FUNCTION_BLOCK PS_PackML_StateMachine_Auto
VAR_INPUT
	Start					:	BOOL;
	Hold					:	BOOL;
	UnHold					:	BOOL;
	Suspend					:	BOOL;
	UnSuspend				:	BOOL;
	Abort					:	BOOL;
	Stop					:	BOOL;
	Complete				:	BOOL;
	Clear					:	BOOL;
	Reset					:	BOOL;
	StateComplete			:	BOOL;
END_VAR
VAR_OUTPUT
	Status					:	WORD;
	// Transient states
	ST_Starting				:	BOOL;
	ST_Completing			:	BOOL;
	ST_Resetting			:	BOOL;
	ST_Holding				:	BOOL;
	ST_UnHolding			:	BOOL;
	ST_Suspending			:	BOOL;
	ST_UnSuspending			:	BOOL;
	ST_Clearing				:	BOOL;
	ST_Stopping				:	BOOL;
	ST_Aborting				:	BOOL;
	// Final states
	ST_Execute				:	BOOL;
	ST_Complete				:	BOOL;
	ST_Idle					:	BOOL;
	ST_Held					:	BOOL;
	ST_Suspended			:	BOOL;
	ST_Stopped				:	BOOL;
	ST_Aborted				:	BOOL;
	
	Error					:	BOOL;
	ErrorID					:	DWORD;
	ePMLState				:	E_PMLState	:=	E_PMLState.IDLE;
END_VAR
VAR
	ePMLStatePrev			:	E_PMLState;
	bStateChange			:	BOOL;
	bStateCompletePrev		:	BOOL;
END_VAR

	// Check for E_PMLState change
	IF ePMLStatePrev <> ePMLState THEN
		ePMLStatePrev	:=	ePMLState;
		bStateChange	:=	TRUE;
	ELSE
		bStateChange	:=	FALSE;
	END_IF
	
	// change to new state if requested
	CASE ePMLState OF
		E_PMLState.UNDEFINED:
			IF bStateChange	THEN
				ST_Starting				:=	FALSE;
				ST_Completing			:=	FALSE;
				ST_Resetting			:=	FALSE;
				ST_Holding				:=	FALSE;
				ST_UnHolding			:=	FALSE;
				ST_Suspending			:=	FALSE;
				ST_UnSuspending			:=	FALSE;
				ST_Clearing				:=	FALSE;
				ST_Stopping				:=	FALSE;
				ST_Aborting				:=	FALSE;
				
				ST_Execute				:=	FALSE;
				ST_Complete				:=	FALSE;
				ST_Idle					:=	FALSE;
				ST_Held					:=	FALSE;
				ST_Suspended			:=	FALSE;
				ST_Stopped				:=	FALSE;
				ST_Aborted				:=	FALSE;
			END_IF
			
			IF Abort THEN
				ePMLState				:=	E_PMLState.ABORTING;
				ST_Aborting				:=	TRUE;
			ELSIF Stop THEN
				ePMLState				:=	E_PMLState.STOPPING;
				ST_Stopping				:=	TRUE;				
			END_IF
		E_PMLState.IDLE:
			IF bStateChange	THEN
				ST_Starting				:=	FALSE;
				ST_Completing			:=	FALSE;
				ST_Resetting			:=	FALSE;
				ST_Holding				:=	FALSE;
				ST_UnHolding			:=	FALSE;
				ST_Suspending			:=	FALSE;
				ST_UnSuspending			:=	FALSE;
				ST_Clearing				:=	FALSE;
				ST_Stopping				:=	FALSE;
				ST_Aborting				:=	FALSE;
				
				ST_Execute				:=	FALSE;
				ST_Complete				:=	FALSE;
				ST_Idle					:=	TRUE;
				ST_Held					:=	FALSE;
				ST_Suspended			:=	FALSE;
				ST_Stopped				:=	FALSE;
				ST_Aborted				:=	FALSE;
			END_IF
			
			IF Abort THEN
				ePMLState				:=	E_PMLState.ABORTING;
				ST_IDLE					:=	FALSE;
				ST_Aborting				:=	TRUE;
			ELSIF Stop THEN
				ePMLState				:=	E_PMLState.STOPPING;
				ST_IDLE					:=	FALSE;
				ST_Stopping				:=	TRUE;
			ELSIF Start THEN
				ePMLState				:=	E_PMLState.STARTING;
				ST_IDLE					:=	FALSE;
				ST_Starting				:=	TRUE;								
			END_IF

		E_PMLState.STARTING:
			IF bStateChange	THEN
				ST_Starting				:=	TRUE;
				ST_Completing			:=	FALSE;
				ST_Resetting			:=	FALSE;
				ST_Holding				:=	FALSE;
				ST_UnHolding			:=	FALSE;
				ST_Suspending			:=	FALSE;
				ST_UnSuspending			:=	FALSE;
				ST_Clearing				:=	FALSE;
				ST_Stopping				:=	FALSE;
				ST_Aborting				:=	FALSE;
				
				ST_Execute				:=	FALSE;
				ST_Complete				:=	FALSE;
				ST_Idle					:=	FALSE;
				ST_Held					:=	FALSE;
				ST_Suspended			:=	FALSE;
				ST_Stopped				:=	FALSE;
				ST_Aborted				:=	FALSE;
			END_IF
			
			IF Abort THEN
				ePMLState				:=	E_PMLState.ABORTING;
				ST_Starting				:=	FALSE;
				ST_Aborting				:=	TRUE;
			ELSIF Stop THEN
				ePMLState				:=	E_PMLState.STOPPING;
				ST_Starting				:=	FALSE;
				ST_Stopping				:=	TRUE;
			ELSIF StateComplete AND NOT bStateCompletePrev THEN
				ePMLState				:=	E_PMLState.EXECUTE;
				bStateCompletePrev		:=	StateComplete;
				ST_Starting				:=	FALSE;
				ST_Execute				:=	TRUE;								
			END_IF

		E_PMLState.EXECUTE:
			IF bStateChange	THEN
				ST_Starting				:=	FALSE;
				ST_Completing			:=	FALSE;
				ST_Resetting			:=	FALSE;
				ST_Holding				:=	FALSE;
				ST_UnHolding			:=	FALSE;
				ST_Suspending			:=	FALSE;
				ST_UnSuspending			:=	FALSE;
				ST_Clearing				:=	FALSE;
				ST_Stopping				:=	FALSE;
				ST_Aborting				:=	FALSE;
				
				ST_Execute				:=	TRUE;
				ST_Complete				:=	FALSE;
				ST_Idle					:=	FALSE;
				ST_Held					:=	FALSE;
				ST_Suspended			:=	FALSE;
				ST_Stopped				:=	FALSE;
				ST_Aborted				:=	FALSE;
			END_IF
			
			IF Abort THEN
				ePMLState				:=	E_PMLState.ABORTING;
				ST_Execute				:=	FALSE;
				ST_Aborting				:=	TRUE;
			ELSIF Stop THEN
				ePMLState				:=	E_PMLState.STOPPING;
				ST_Execute				:=	FALSE;
				ST_Stopping				:=	TRUE;
			ELSIF Hold THEN
				ePMLState				:=	E_PMLState.HOLDING;
				ST_Execute				:=	FALSE;
				ST_Holding				:=	TRUE;
			ELSIF Suspend THEN
				ePMLState				:=	E_PMLState.SUSPENDING;
				ST_Execute				:=	FALSE;
				ST_Suspending			:=	TRUE;
			ELSIF Complete THEN
				ePMLState				:=	E_PMLState.COMPLETING;
				ST_Execute				:=	FALSE;
				ST_Completing			:=	TRUE;	
			END_IF

		E_PMLState.COMPLETING:
			IF bStateChange	THEN
				ST_Starting				:=	FALSE;
				ST_Completing			:=	TRUE;
				ST_Resetting			:=	FALSE;
				ST_Holding				:=	FALSE;
				ST_UnHolding			:=	FALSE;
				ST_Suspending			:=	FALSE;
				ST_UnSuspending			:=	FALSE;
				ST_Clearing				:=	FALSE;
				ST_Stopping				:=	FALSE;
				ST_Aborting				:=	FALSE;
				
				ST_Execute				:=	FALSE;
				ST_Complete				:=	FALSE;
				ST_Idle					:=	FALSE;
				ST_Held					:=	FALSE;
				ST_Suspended			:=	FALSE;
				ST_Stopped				:=	FALSE;
				ST_Aborted				:=	FALSE;
			END_IF
			
			IF Abort THEN
				ePMLState				:=	E_PMLState.ABORTING;
				ST_Completing			:=	FALSE;
				ST_Aborting				:=	TRUE;
			ELSIF Stop THEN
				ePMLState				:=	E_PMLState.STOPPING;
				ST_Completing			:=	FALSE;
				ST_Stopping				:=	TRUE;
			ELSIF StateComplete AND NOT bStateCompletePrev THEN
				ePMLState				:=	E_PMLState.COMPLETE;
				bStateCompletePrev		:=	StateComplete;
				ST_Completing			:=	FALSE;
				ST_Complete				:=	TRUE;								
			END_IF
			
		E_PMLState.COMPLETE:
			IF bStateChange	THEN
				ST_Starting				:=	FALSE;
				ST_Completing			:=	FALSE;
				ST_Resetting			:=	FALSE;
				ST_Holding				:=	FALSE;
				ST_UnHolding			:=	FALSE;
				ST_Suspending			:=	FALSE;
				ST_UnSuspending			:=	FALSE;
				ST_Clearing				:=	FALSE;
				ST_Stopping				:=	FALSE;
				ST_Aborting				:=	FALSE;
				
				ST_Execute				:=	FALSE;
				ST_Complete				:=	TRUE;
				ST_Idle					:=	FALSE;
				ST_Held					:=	FALSE;
				ST_Suspended			:=	FALSE;
				ST_Stopped				:=	FALSE;
				ST_Aborted				:=	FALSE;
			END_IF
			
			IF Abort THEN
				ePMLState				:=	E_PMLState.ABORTING;
				ST_Complete				:=	FALSE;
				ST_Aborting				:=	TRUE;
			ELSIF Stop THEN
				ePMLState				:=	E_PMLState.STOPPING;
				ST_Complete				:=	FALSE;
				ST_Stopping				:=	TRUE;
			ELSIF Reset THEN
				ePMLState				:=	E_PMLState.RESETTING;
				ST_Complete				:=	FALSE;
				ST_Resetting			:=	TRUE;
			END_IF

		E_PMLState.RESETTING:
			IF bStateChange	THEN
				ST_Starting				:=	FALSE;
				ST_Completing			:=	FALSE;
				ST_Resetting			:=	TRUE;
				ST_Holding				:=	FALSE;
				ST_UnHolding			:=	FALSE;
				ST_Suspending			:=	FALSE;
				ST_UnSuspending			:=	FALSE;
				ST_Clearing				:=	FALSE;
				ST_Stopping				:=	FALSE;
				ST_Aborting				:=	FALSE;
				
				ST_Execute				:=	FALSE;
				ST_Complete				:=	FALSE;
				ST_Idle					:=	FALSE;
				ST_Held					:=	FALSE;
				ST_Suspended			:=	FALSE;
				ST_Stopped				:=	FALSE;
				ST_Aborted				:=	FALSE;
			END_IF
			
			IF Abort THEN
				ePMLState				:=	E_PMLState.ABORTING;
				ST_Resetting			:=	FALSE;
				ST_Aborting				:=	TRUE;
			ELSIF Stop THEN
				ePMLState				:=	E_PMLState.STOPPING;
				ST_Resetting			:=	FALSE;
				ST_Stopping				:=	TRUE;
			ELSIF StateComplete AND NOT bStateCompletePrev THEN
				ePMLState				:=	E_PMLState.IDLE;
				bStateCompletePrev		:=	StateComplete;
				ST_Resetting			:=	FALSE;
				ST_Idle					:=	TRUE;								
			END_IF
		
		E_PMLState.HOLDING:
			IF bStateChange	THEN
				ST_Starting				:=	FALSE;
				ST_Completing			:=	FALSE;
				ST_Resetting			:=	FALSE;
				ST_Holding				:=	TRUE;
				ST_UnHolding			:=	FALSE;
				ST_Suspending			:=	FALSE;
				ST_UnSuspending			:=	FALSE;
				ST_Clearing				:=	FALSE;
				ST_Stopping				:=	FALSE;
				ST_Aborting				:=	FALSE;
				
				ST_Execute				:=	FALSE;
				ST_Complete				:=	FALSE;
				ST_Idle					:=	FALSE;
				ST_Held					:=	FALSE;
				ST_Suspended			:=	FALSE;
				ST_Stopped				:=	FALSE;
				ST_Aborted				:=	FALSE;
			END_IF
			
			IF Abort THEN
				ePMLState				:=	E_PMLState.ABORTING;
				ST_Holding				:=	FALSE;
				ST_Aborting				:=	TRUE;
			ELSIF Stop THEN
				ePMLState				:=	E_PMLState.STOPPING;
				ST_Holding				:=	FALSE;
				ST_Stopping				:=	TRUE;
			ELSIF StateComplete AND NOT bStateCompletePrev THEN
				ePMLState				:=	E_PMLState.HELD;
				bStateCompletePrev		:=	StateComplete;
				ST_Holding				:=	FALSE;
				ST_Held					:=	TRUE;								
			END_IF
			
		E_PMLState.HELD:
			IF bStateChange	THEN
				ST_Starting				:=	FALSE;
				ST_Completing			:=	FALSE;
				ST_Resetting			:=	FALSE;
				ST_Holding				:=	FALSE;
				ST_UnHolding			:=	FALSE;
				ST_Suspending			:=	FALSE;
				ST_UnSuspending			:=	FALSE;
				ST_Clearing				:=	FALSE;
				ST_Stopping				:=	FALSE;
				ST_Aborting				:=	FALSE;
				
				ST_Execute				:=	FALSE;
				ST_Complete				:=	FALSE;
				ST_Idle					:=	FALSE;
				ST_Held					:=	TRUE;
				ST_Suspended			:=	FALSE;
				ST_Stopped				:=	FALSE;
				ST_Aborted				:=	FALSE;
			END_IF
			
			IF Abort THEN
				ePMLState				:=	E_PMLState.ABORTING;
				ST_Held					:=	FALSE;
				ST_Aborting				:=	TRUE;
			ELSIF Stop THEN
				ePMLState				:=	E_PMLState.STOPPING;
				ST_Held					:=	FALSE;
				ST_Stopping				:=	TRUE;
			ELSIF UnHold THEN
				ePMLState				:=	E_PMLState.UNHOLDING;
				ST_Held					:=	FALSE;
				ST_UnHolding			:=	TRUE;
			END_IF

		E_PMLState.UNHOLDING:	
			IF bStateChange	THEN
				ST_Starting				:=	FALSE;
				ST_Completing			:=	FALSE;
				ST_Resetting			:=	FALSE;
				ST_Holding				:=	FALSE;
				ST_UnHolding			:=	TRUE;
				ST_Suspending			:=	FALSE;
				ST_UnSuspending			:=	FALSE;
				ST_Clearing				:=	FALSE;
				ST_Stopping				:=	FALSE;
				ST_Aborting				:=	FALSE;
				
				ST_Execute				:=	FALSE;
				ST_Complete				:=	FALSE;
				ST_Idle					:=	FALSE;
				ST_Held					:=	FALSE;
				ST_Suspended			:=	FALSE;
				ST_Stopped				:=	FALSE;
				ST_Aborted				:=	FALSE;
			END_IF
			
			IF Abort THEN
				ePMLState				:=	E_PMLState.ABORTING;
				ST_UnHolding			:=	FALSE;
				ST_Aborting				:=	TRUE;
			ELSIF Stop THEN
				ePMLState				:=	E_PMLState.STOPPING;
				ST_UnHolding			:=	FALSE;
				ST_Stopping				:=	TRUE;
			ELSIF StateComplete AND NOT bStateCompletePrev THEN
				ePMLState				:=	E_PMLState.EXECUTE;
				bStateCompletePrev		:=	StateComplete;
				ST_UnHolding			:=	FALSE;
				ST_Execute				:=	TRUE;								
			END_IF
			
		E_PMLState.SUSPENDING:
			IF bStateChange	THEN
				ST_Starting				:=	FALSE;
				ST_Completing			:=	FALSE;
				ST_Resetting			:=	FALSE;
				ST_Holding				:=	FALSE;
				ST_UnHolding			:=	FALSE;
				ST_Suspending			:=	TRUE;
				ST_UnSuspending			:=	FALSE;
				ST_Clearing				:=	FALSE;
				ST_Stopping				:=	FALSE;
				ST_Aborting				:=	FALSE;
				
				ST_Execute				:=	FALSE;
				ST_Complete				:=	FALSE;
				ST_Idle					:=	FALSE;
				ST_Held					:=	FALSE;
				ST_Suspended			:=	FALSE;
				ST_Stopped				:=	FALSE;
				ST_Aborted				:=	FALSE;
			END_IF
			
			IF Abort THEN
				ePMLState				:=	E_PMLState.ABORTING;
				ST_Suspending			:=	FALSE;
				ST_Aborting				:=	TRUE;
			ELSIF Stop THEN
				ePMLState				:=	E_PMLState.STOPPING;
				ST_Suspending			:=	FALSE;
				ST_Stopping				:=	TRUE;
			ELSIF StateComplete AND NOT bStateCompletePrev THEN
				ePMLState				:=	E_PMLState.SUSPENDED;
				bStateCompletePrev		:=	StateComplete;
				ST_Suspending			:=	FALSE;
				ST_Suspended			:=	TRUE;								
			END_IF
		
		E_PMLState.SUSPENDED:
			IF bStateChange	THEN
				ST_Starting				:=	FALSE;
				ST_Completing			:=	FALSE;
				ST_Resetting			:=	FALSE;
				ST_Holding				:=	FALSE;
				ST_UnHolding			:=	FALSE;
				ST_Suspending			:=	FALSE;
				ST_UnSuspending			:=	FALSE;
				ST_Clearing				:=	FALSE;
				ST_Stopping				:=	FALSE;
				ST_Aborting				:=	FALSE;
				
				ST_Execute				:=	FALSE;
				ST_Complete				:=	FALSE;
				ST_Idle					:=	FALSE;
				ST_Held					:=	FALSE;
				ST_Suspended			:=	TRUE;
				ST_Stopped				:=	FALSE;
				ST_Aborted				:=	FALSE;
			END_IF
			
			IF Abort THEN
				ePMLState				:=	E_PMLState.ABORTING;
				ST_Suspended			:=	FALSE;
				ST_Aborting				:=	TRUE;
			ELSIF Stop THEN
				ePMLState				:=	E_PMLState.STOPPING;
				ST_Suspended			:=	FALSE;
				ST_Stopping				:=	TRUE;
			ELSIF UnSuspend THEN
				ePMLState				:=	E_PMLState.UNSUSPENDING;
				ST_Suspended			:=	FALSE;
				ST_UnSuspending			:=	TRUE;
			END_IF

		E_PMLState.UNSUSPENDING:	
			IF bStateChange	THEN
				ST_Starting				:=	FALSE;
				ST_Completing			:=	FALSE;
				ST_Resetting			:=	FALSE;
				ST_Holding				:=	FALSE;
				ST_UnHolding			:=	FALSE;
				ST_Suspending			:=	FALSE;
				ST_UnSuspending			:=	TRUE;
				ST_Clearing				:=	FALSE;
				ST_Stopping				:=	FALSE;
				ST_Aborting				:=	FALSE;
				
				ST_Execute				:=	FALSE;
				ST_Complete				:=	FALSE;
				ST_Idle					:=	FALSE;
				ST_Held					:=	FALSE;
				ST_Suspended			:=	FALSE;
				ST_Stopped				:=	FALSE;
				ST_Aborted				:=	FALSE;
			END_IF
			
			IF Abort THEN
				ePMLState				:=	E_PMLState.ABORTING;
				ST_UnSuspending			:=	FALSE;
				ST_Aborting				:=	TRUE;
			ELSIF Stop THEN
				ePMLState				:=	E_PMLState.STOPPING;
				ST_UnSuspending			:=	FALSE;
				ST_Stopping				:=	TRUE;
			ELSIF StateComplete AND NOT bStateCompletePrev THEN
				ePMLState				:=	E_PMLState.EXECUTE;
				bStateCompletePrev		:=	StateComplete;
				ST_UnSuspending			:=	FALSE;
				ST_Execute				:=	TRUE;								
			END_IF
		
		E_PMLState.STOPPING:
			IF bStateChange	THEN
				ST_Starting				:=	FALSE;
				ST_Completing			:=	FALSE;
				ST_Resetting			:=	FALSE;
				ST_Holding				:=	FALSE;
				ST_UnHolding			:=	FALSE;
				ST_Suspending			:=	FALSE;
				ST_UnSuspending			:=	FALSE;
				ST_Clearing				:=	FALSE;
				ST_Stopping				:=	TRUE;
				ST_Aborting				:=	FALSE;
				
				ST_Execute				:=	FALSE;
				ST_Complete				:=	FALSE;
				ST_Idle					:=	FALSE;
				ST_Held					:=	FALSE;
				ST_Suspended			:=	FALSE;
				ST_Stopped				:=	FALSE;
				ST_Aborted				:=	FALSE;
			END_IF
			
			IF Abort THEN
				ePMLState				:=	E_PMLState.ABORTING;
				ST_Stopping				:=	FALSE;
				ST_Aborting				:=	TRUE;
			ELSIF StateComplete AND NOT bStateCompletePrev THEN
				ePMLState				:=	E_PMLState.STOPPED;
				bStateCompletePrev		:=	StateComplete;
				ST_Stopping				:=	FALSE;
				ST_Stopped				:=	TRUE;								
			END_IF

		E_PMLState.STOPPED:
			IF bStateChange	THEN
				ST_Starting				:=	FALSE;
				ST_Completing			:=	FALSE;
				ST_Resetting			:=	FALSE;
				ST_Holding				:=	FALSE;
				ST_UnHolding			:=	FALSE;
				ST_Suspending			:=	FALSE;
				ST_UnSuspending			:=	FALSE;
				ST_Clearing				:=	FALSE;
				ST_Stopping				:=	FALSE;
				ST_Aborting				:=	FALSE;
				
				ST_Execute				:=	FALSE;
				ST_Complete				:=	FALSE;
				ST_Idle					:=	FALSE;
				ST_Held					:=	FALSE;
				ST_Suspended			:=	FALSE;
				ST_Stopped				:=	TRUE;
				ST_Aborted				:=	FALSE;
			END_IF
			
			IF Abort THEN
				ePMLState				:=	E_PMLState.ABORTING;
				ST_Stopped				:=	FALSE;
				ST_Aborting				:=	TRUE;
			ELSIF Reset THEN
				ePMLState				:=	E_PMLState.RESETTING;
				ST_Stopped				:=	FALSE;
				ST_Resetting			:=	TRUE;
			END_IF
		
		E_PMLState.ABORTING:
			IF bStateChange	THEN
				ST_Starting				:=	FALSE;
				ST_Completing			:=	FALSE;
				ST_Resetting			:=	FALSE;
				ST_Holding				:=	FALSE;
				ST_UnHolding			:=	FALSE;
				ST_Suspending			:=	FALSE;
				ST_UnSuspending			:=	FALSE;
				ST_Clearing				:=	FALSE;
				ST_Stopping				:=	FALSE;
				ST_Aborting				:=	TRUE;
				
				ST_Execute				:=	FALSE;
				ST_Complete				:=	FALSE;
				ST_Idle					:=	FALSE;
				ST_Held					:=	FALSE;
				ST_Suspended			:=	FALSE;
				ST_Stopped				:=	FALSE;
				ST_Aborted				:=	FALSE;
			END_IF
			
			IF StateComplete AND NOT bStateCompletePrev THEN
				ePMLState				:=	E_PMLState.ABORTED;
				bStateCompletePrev		:=	StateComplete;
				ST_Aborting				:=	FALSE;
				ST_Aborted				:=	TRUE;								
			END_IF
			
		E_PMLState.ABORTED:
			IF bStateChange	THEN
				ST_Starting				:=	FALSE;
				ST_Completing			:=	FALSE;
				ST_Resetting			:=	FALSE;
				ST_Holding				:=	FALSE;
				ST_UnHolding			:=	FALSE;
				ST_Suspending			:=	FALSE;
				ST_UnSuspending			:=	FALSE;
				ST_Clearing				:=	FALSE;
				ST_Stopping				:=	FALSE;
				ST_Aborting				:=	FALSE;
				
				ST_Execute				:=	FALSE;
				ST_Complete				:=	FALSE;
				ST_Idle					:=	FALSE;
				ST_Held					:=	FALSE;
				ST_Suspended			:=	FALSE;
				ST_Stopped				:=	FALSE;
				ST_Aborted				:=	TRUE;
			END_IF
			
			IF Clear THEN
				ePMLState				:=	E_PMLState.CLEARING;
				ST_Aborted				:=	FALSE;
				ST_Clearing				:=	TRUE;
			END_IF
		
		E_PMLState.CLEARING:
			IF bStateChange	THEN
				ST_Starting				:=	FALSE;
				ST_Completing			:=	FALSE;
				ST_Resetting			:=	FALSE;
				ST_Holding				:=	FALSE;
				ST_UnHolding			:=	FALSE;
				ST_Suspending			:=	FALSE;
				ST_UnSuspending			:=	FALSE;
				ST_Clearing				:=	TRUE;
				ST_Stopping				:=	FALSE;
				ST_Aborting				:=	FALSE;
				
				ST_Execute				:=	FALSE;
				ST_Complete				:=	FALSE;
				ST_Idle					:=	FALSE;
				ST_Held					:=	FALSE;
				ST_Suspended			:=	FALSE;
				ST_Stopped				:=	FALSE;
				ST_Aborted				:=	FALSE;
			END_IF
			
			IF Abort THEN
				ePMLState				:=	E_PMLState.ABORTING;
				ST_Clearing				:=	FALSE;
				ST_Aborting				:=	TRUE;
			ELSIF Stop THEN
				ePMLState				:=	E_PMLState.STOPPING;
				ST_Clearing				:=	FALSE;
				ST_Stopping				:=	TRUE;
			ELSIF StateComplete AND NOT bStateCompletePrev THEN
				ePMLState				:=	E_PMLState.STOPPED;
				bStateCompletePrev		:=	StateComplete;
				ST_Clearing				:=	FALSE;
				ST_Stopped				:=	TRUE;								
			END_IF
		
	END_CASE
	
	// bStateCompletePrev := bStateCompletePrev AND StateComplete;

END_FUNCTION_BLOCK

(* stored: Version 1.1.0.1, ProductVersion 3.1.4024.15
   POU PS_PackML_StateMachine_Auto: Id {3668b145-0585-4c98-8643-0094daaebffe}, SpecialFunc None *)
